// TIA Portal project "Silosteuerung" (V15)

(* hardware
DEVICE "S7-1200-Station_1"  S7-1200 Station
   slot 0: "Baugruppenträger_0"  S7-1200 Rack  Rack  V1.0
   slot 1: "PLC_1"  CPU 1214C DC/DC/Rly  6ES7 214-1HG40-0XB0  V4.2
*)

// ===== PLC "PLC_1"  CPU 1214C DC/DC/Rly =====

VAR_GLOBAL   // PLC tag table "Standard-Variablentabelle"
   "Clock_Byte" AT %MB100 : Byte;
   "Clock_10Hz" AT %M100.0 : Bool;
   "Clock_5Hz" AT %M100.1 : Bool;
   "Clock_2.5Hz" AT %M100.2 : Bool;
   "Clock_2Hz" AT %M100.3 : Bool;
   "Clock_1.25Hz" AT %M100.4 : Bool;
   "Clock_1Hz" AT %M100.5 : Bool;
   "Clock_0.625Hz" AT %M100.6 : Bool;
   "Clock_0.5Hz" AT %M100.7 : Bool;
   "S0" AT %I0.0 : Bool;   // Aus Taster
   "S1" AT %I0.1 : Bool;   // Ein Taster
   "S2" AT %I0.2 : Bool;   // Not-Halt
   "S3" AT %I0.3 : Bool;   // Stop-Befüllen
   "S4" AT %I0.4 : Bool;   // Start-Befüllen
   "S5" AT %I0.5 : Bool;   // Lampen-Kontrolle
   "S6" AT %I0.6 : Bool;   // Störung Quittieren/ Reset Not-Halt
   "S10" AT %I0.7 : Bool;   // Wagen vorhanden
   "S11" AT %I1.0 : Bool;   // Wagen voll
   "Q3" AT %I1.1 : Bool;   // Motorschutzschalter (MSS)
   "P1" AT %Q0.0 : Bool;   // Anlage Ein
   "P2" AT %Q0.1 : Bool;   // Anlage Sammelstörung
   "P3" AT %Q0.2 : Bool;   // Motor Förderband
   "P4" AT %Q0.3 : Bool;   // Wagen vorhanden
   "P5" AT %Q0.4 : Bool;   // Wagen voll
   "P6" AT %Q0.5 : Bool;   // Magnetventil Y1 ein
   "P7" AT %Q0.6 : Bool;   // Schneckenförderer ein
   "T7" AT %Q0.7 : Bool;   // Freigabe Schneckenförderer
   "Q1" AT %Q1.0 : Bool;   // Freigabe Förderband
   "Merker Anlage Betriebsbereit" AT %M10.1 : Bool;
   "Merker Anlage Befüllen" AT %M10.2 : Bool;
   "Merker Schneckenförderer" AT %M10.3 : Bool;
   "Merker Störung MSS" AT %M10.4 : Bool;
   "Merker Lampentest" AT %M10.5 : Bool;
   "Merker Not-Halt-Störung" AT %M10.6 : Bool;
   "Füllstand AI" AT %IW64 : Word;
END_VAR

DATA_BLOCK "Analogwertverarbeitung"   // DB3
{ S7_Optimized_Access := 'TRUE' }
VERSION : 0.1
   VAR
      "Analogwert Normieren" : Real;
      "Analogwert Skalieren" : Real;
   END_VAR
BEGIN
END_DATA_BLOCK

// folder: System blocks/Program resources

DATA_BLOCK "IEC_Timer_0_DB_10"   // DB12
{ S7_Optimized_Access := 'TRUE' }
AUTHOR : Simatic
FAMILY : IEC
NAME : IEC_TMR
VERSION : 1.0
// stored: InstanceOfName IEC_TIMER
"IEC_TIMER"
BEGIN
END_DATA_BLOCK

DATA_BLOCK "IEC_Timer_0_DB_11"   // DB13
{ S7_Optimized_Access := 'TRUE' }
AUTHOR : Simatic
FAMILY : IEC
NAME : IEC_TMR
VERSION : 1.0
// stored: InstanceOfName IEC_TIMER
"IEC_TIMER"
BEGIN
END_DATA_BLOCK

// folder: (top level)

FUNCTION "Silosteuerung" : Void   // FC1, FBD
TITLE = Silosteuerung
{ S7_Optimized_Access := 'TRUE' }
VERSION : 0.1
BEGIN

REGION Network 1: Anlage Ein
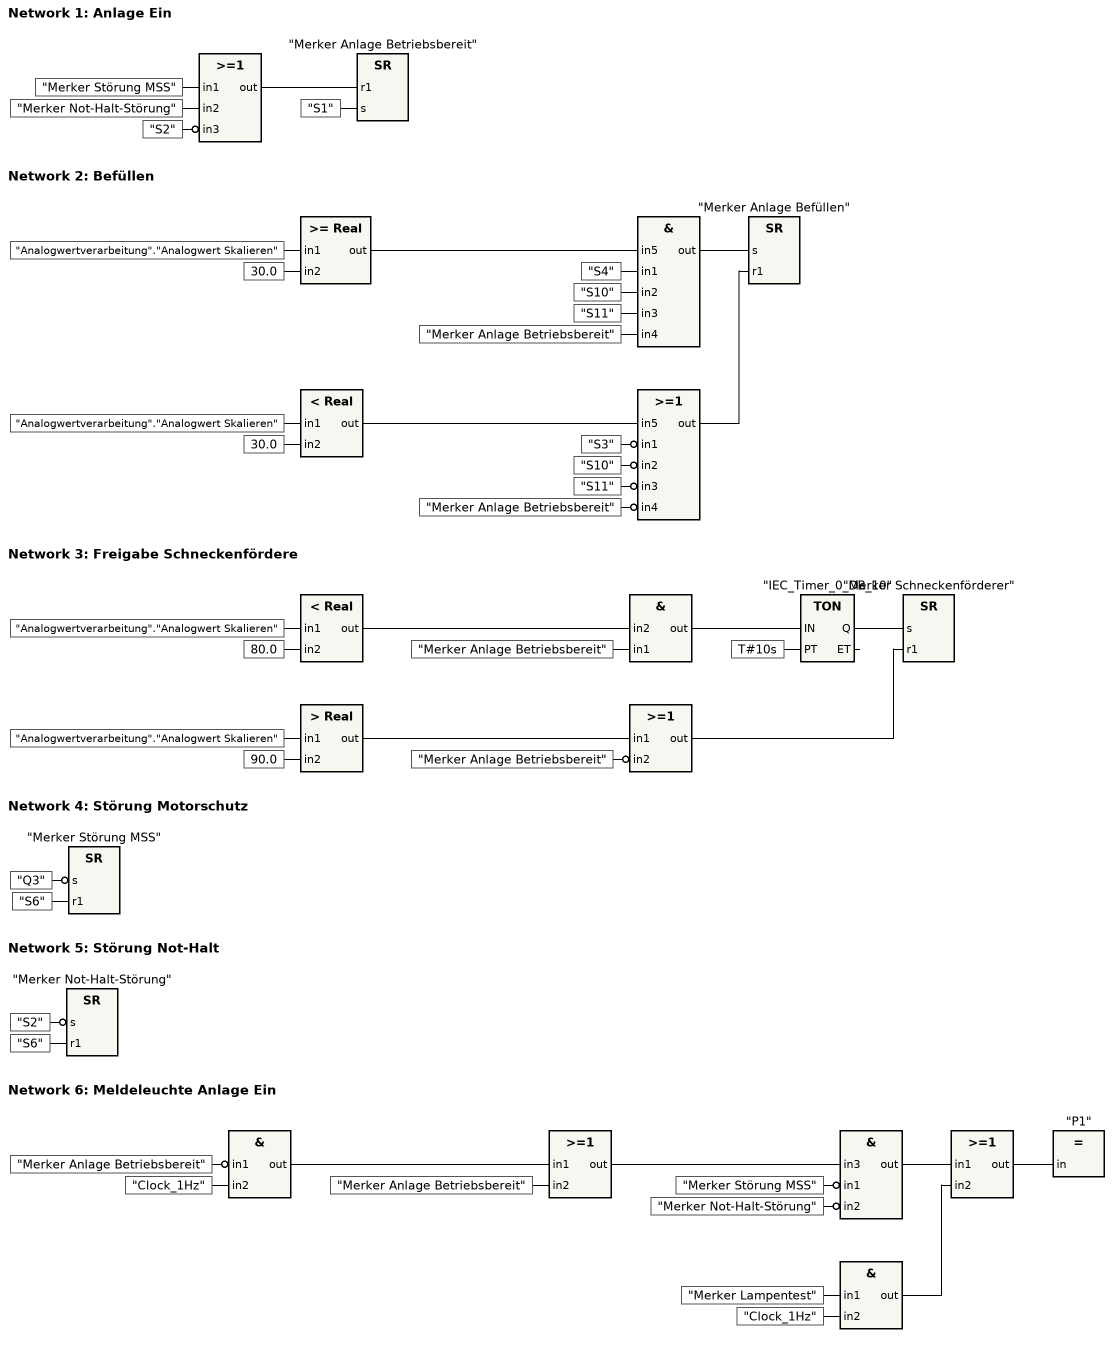
   IF "S1" THEN
       "Merker Anlage Betriebsbereit" := TRUE;   // SR flip-flop
   END_IF;
   IF "Merker Störung MSS" OR "Merker Not-Halt-Störung" OR NOT "S2" THEN
       "Merker Anlage Betriebsbereit" := FALSE;
   END_IF;
END_REGION

REGION Network 2: Befüllen
   IF ("Analogwertverarbeitung"."Analogwert Skalieren" >= 30.0) AND "S4" AND "S10" AND "S11" AND "Merker Anlage Betriebsbereit" THEN
       "Merker Anlage Befüllen" := TRUE;   // SR flip-flop
   END_IF;
   IF ("Analogwertverarbeitung"."Analogwert Skalieren" < 30.0) OR NOT "S3" OR NOT "S10" OR NOT "S11" OR NOT "Merker Anlage Betriebsbereit" THEN
       "Merker Anlage Befüllen" := FALSE;
   END_IF;
END_REGION

REGION Network 3: Freigabe Schneckenfördere
   "IEC_Timer_0_DB_10".TON(IN := ("Analogwertverarbeitung"."Analogwert Skalieren" < 80.0) AND "Merker Anlage Betriebsbereit",
                           PT := T#10s);
   IF "IEC_Timer_0_DB_10".Q THEN
       "Merker Schneckenförderer" := TRUE;   // SR flip-flop
   END_IF;
   IF ("Analogwertverarbeitung"."Analogwert Skalieren" > 90.0) OR NOT "Merker Anlage Betriebsbereit" THEN
       "Merker Schneckenförderer" := FALSE;
   END_IF;
END_REGION

REGION Network 4: Störung Motorschutz
   IF NOT "Q3" THEN
       "Merker Störung MSS" := TRUE;   // SR flip-flop
   END_IF;
   IF "S6" THEN "Merker Störung MSS" := FALSE; END_IF;
END_REGION

REGION Network 5: Störung Not-Halt
   IF NOT "S2" THEN
       "Merker Not-Halt-Störung" := TRUE;   // SR flip-flop
   END_IF;
   IF "S6" THEN "Merker Not-Halt-Störung" := FALSE; END_IF;
END_REGION

REGION Network 6: Meldeleuchte Anlage Ein
   "P1" := (((NOT "Merker Anlage Betriebsbereit" AND "Clock_1Hz") OR "Merker Anlage Betriebsbereit") AND NOT "Merker Störung MSS" AND NOT "Merker Not-Halt-Störung") OR ("Merker Lampentest" AND "Clock_1Hz");
END_REGION

REGION Network 7: Sammelstörung
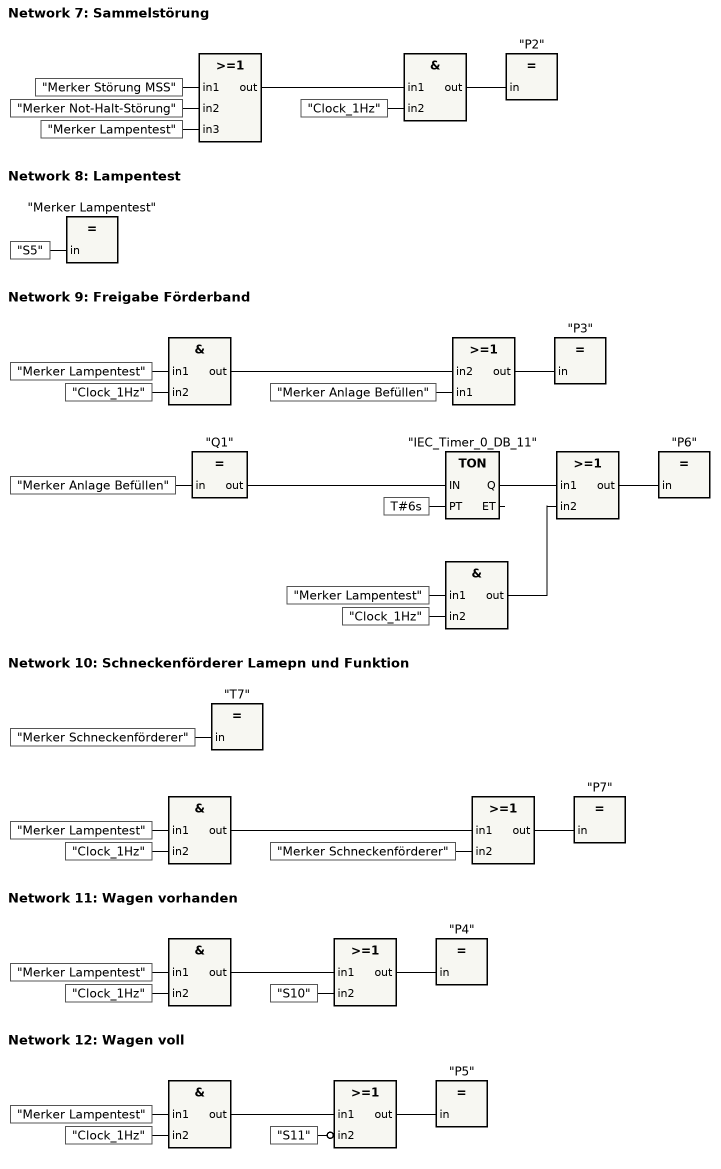
   "P2" := ("Merker Störung MSS" OR "Merker Not-Halt-Störung" OR "Merker Lampentest") AND "Clock_1Hz";
END_REGION

REGION Network 8: Lampentest
   "Merker Lampentest" := "S5";
END_REGION

REGION Network 9: Freigabe Förderband
   "P3" := ("Merker Lampentest" AND "Clock_1Hz") OR "Merker Anlage Befüllen";
   "Q1" := "Merker Anlage Befüllen";
   "IEC_Timer_0_DB_11".TON(IN := "Merker Anlage Befüllen", PT := T#6s);
   "P6" := "IEC_Timer_0_DB_11".Q OR ("Merker Lampentest" AND "Clock_1Hz");
END_REGION

REGION Network 10: Schneckenförderer Lamepn und Funktion
   "T7" := "Merker Schneckenförderer";
   "P7" := ("Merker Lampentest" AND "Clock_1Hz") OR "Merker Schneckenförderer";
END_REGION

REGION Network 11: Wagen vorhanden
   "P4" := ("Merker Lampentest" AND "Clock_1Hz") OR "S10";
END_REGION

REGION Network 12: Wagen voll
   "P5" := ("Merker Lampentest" AND "Clock_1Hz") OR NOT "S11";
END_REGION

REGION Network 13
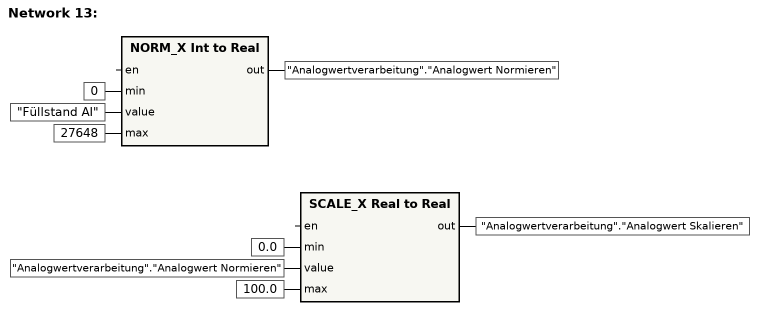
   "Analogwertverarbeitung"."Analogwert Normieren" := NORM_X(MIN := 0, VALUE := "Füllstand AI", MAX := 27648);
   "Analogwertverarbeitung"."Analogwert Skalieren" := SCALE_X(MIN := 0.0, VALUE := "Analogwertverarbeitung"."Analogwert Normieren", MAX := 100.0);
END_REGION
END_FUNCTION

ORGANIZATION_BLOCK "Main"   // OB1, LAD, ProgramCycle
TITLE = "Main Program Sweep (Cycle)"
{ S7_Optimized_Access := 'TRUE' }
VERSION : 0.1
   VAR_INPUT
      Initial_Call : Bool;   // Initial call of this OB
      Remanence : Bool;   // =True, if remanent data are available
   END_VAR
BEGIN

REGION Network 1
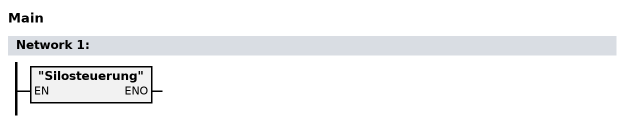
   RUNG wire#powerrail
      "Silosteuerung"()
   END_RUNG
   // the same network as SCL:
   "Silosteuerung"();
END_REGION
END_ORGANIZATION_BLOCK